(* PLC project Tc2_System.F_GetStructMemberAlignment Demo, tc3-libraries-kb TwinCAT 3.1 *)
(* stored: creationDateTime 2026-05-20T00:00:00, modificationDateTime 2026-05-20T00:00:00 *)

PROGRAM P_Demo_F_GetStructMemberAlignment
  VAR
    nAlignBytes : BYTE;  (* 当前平台对齐字节数（1 / 2 / 4 / 8） *)
  END_VAR

// =============================================================================
// 场景：启动时记录当前平台对齐字节数到全局诊断变量；跨平台部署时一眼看出差异。
// 价值：实测最准，替代凭经验猜。
// 验证：在 x86 工控机上观察 nAlignBytes = 8；在 Arm CX 上观察 = 4。
// 验证步骤：
//   1. 右键 PLC 项目 → Import PLCopenXML → 选本文件
//   2. 引用 Tc2_System（References → Add library）
//   3. 编译 → 登录 → 运行；按上方『验证』行的指示在线写值观察
// =============================================================================

// 一次调用即可，平台对齐不会运行期改变
nAlignBytes := F_GetStructMemberAlignment();
END_PROGRAM
